{attribute 'Tc2GvlVarNames'}
VAR_GLOBAL

FE_Bp_arus			:F_TRIG;
RE_Bp_dcy			:R_TRIG;
Joystick			:BOOL;	//Au moins 1 direction actionnée

Cde_Desserrage_presseurs			:		BOOL;
Cde_Serrage_Presseurs				:		BOOL;

Cmd_SerDes_Pince:BOOL;

Cde_Serr_Clamps	:BOOL;
Cde_Dess_Clamps	:BOOL;


END_VAR

(* stored: Version 1.1.0.1, ProductVersion 3.1.4024.15
   GVL Global_Commandes: Id {52054f80-4379-4cf9-9ee7-a53a6fbb8b5c} *)
